{attribute 'qualified_only'}
VAR_GLOBAL RETAIN
	ChargerDelay_TON : ARRAY[1..6] OF TON;
	ChargerDelay_PT  : ARRAY[1..6] OF TIME;
	ChargerDelay_ET  : ARRAY[1..6] OF TIME;	
	
	LongestChargeTime_TON : TON;
	LongestChargeTime_PT : TIME;
	LongestChargeTime_ET : TIME;

	ChargeTimeStartDelay	: ARRAY[1..6] OF INT;
	ChargingTimeElapse		: ARRAY[1..6] OF INT;	
	ChargingTimeElapse_TON	: ARRAY[1..6] OF TON;
	
	//sending the longest charge time elaps to P1 PP HMI
	EchoLongestChargerTimeDelay  : INT;
	EchoLongestChargerTimeElapse : INT;	

END_VAR

(* stored: Version 1.1.0.1, ProductVersion 3.1.4024.11
   GVL ChargeTime_DB: Id {aef6f516-ebaa-4401-acff-5fe912a2763d} *)
